Staubli VAL3: exeSA.pgx

program exeSA(dio x_dInput, dio x_dOutput, num x_nLength)
begin

  while true
    x_dOutput=true
    wait(x_dInput==false)
    if (!watch(x_dInput==true,x_nLength))
      x_dOutput=false
    endIf
    wait(x_dInput==true)
    x_dOutput=true
  endWhile
end
